FUNCTION_BLOCK AddPermitter (* Composite Function Block Type *)
  (* Standard: 61499-2 *)
  (* Version 0.0, 10/19/2017, chivdan, nxtControl GmbH, template *)
  PACKAGE Main;
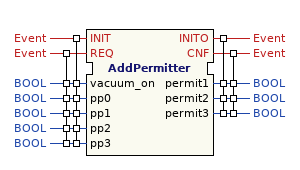
  EVENT_INPUT
    INIT WITH vacuum_on, pp0, pp1, pp2, pp3; (* Initialization Request *)
    REQ WITH vacuum_on, pp0, pp1, pp2, pp3;
  END_EVENT
  EVENT_OUTPUT
    INITO WITH permit1, permit2, permit3; (* Initialization Confirm *)
    CNF WITH permit1, permit2, permit3; (* Execution Confirmation *)
  END_EVENT
  VAR_INPUT
    vacuum_on : BOOL; (* Input event qualifier *)
    pp0 : BOOL;
    pp1 : BOOL;
    pp2 : BOOL;
    pp3 : BOOL;
  END_VAR
  VAR_OUTPUT
    permit1 : BOOL; (* Output event qualifier *)
    permit2 : BOOL;
    permit3 : BOOL;
  END_VAR
  FBS
    WP1 : pickup;
    WP2 : pickup;
    WP3 : pickup;
    FB1 : RandomAddSupplier;
    FB2 : AND_EVENTS;
    FB3 : AND_-2118623424; {SET_ATTRIBUTE(Configuration.GenericFBType.InterfaceParams, Runtime.Standard#CNT:=2;OUT:BOOL)}
    FB4 : AND_EVENTS;
    FB5 : AND_-2118623424; {SET_ATTRIBUTE(Configuration.GenericFBType.InterfaceParams, Runtime.Standard#CNT:=2;OUT:BOOL)}
    FB6 : AND_EVENTS;
    FB7 : AND_-2118623424; {SET_ATTRIBUTE(Configuration.GenericFBType.InterfaceParams, Runtime.Standard#CNT:=2;OUT:BOOL)}
    FB8 : E_MERGE;
    FB9 : E_MERGE;
  END_FBS
  EVENT_CONNECTIONS
    INIT TO WP1.INIT;
    WP1.INITO TO WP2.INIT;
    WP2.INITO TO WP3.INIT;
    WP3.INITO TO INITO;
    INIT TO FB1.INIT;
    FB2.CNF TO FB3.REQ;
    WP1.CNF TO FB2.MODEL;
    FB1.CNF TO FB2.ADDER;
    FB1.CNF TO FB4.ADDER;
    FB1.CNF TO FB6.ADDER;
    WP2.CNF TO FB4.MODEL;
    WP3.CNF TO FB6.MODEL;
    FB4.CNF TO FB5.REQ;
    FB6.CNF TO FB7.REQ;
    FB3.CNF TO FB8.EI1;
    FB5.CNF TO FB8.EI2;
    FB8.EO TO FB9.EI1;
    FB7.CNF TO FB9.EI2;
    FB9.EO TO CNF;
    REQ TO WP1.REQ;
    REQ TO WP2.REQ;
    REQ TO WP3.REQ;
  END_CONNECTIONS
  DATA_CONNECTIONS
    vacuum_on TO WP1.vacuum_on;
    pp1 TO WP1.pp;
    pp2 TO WP2.pp;
    pp3 TO WP3.pp;
    pp0 TO WP1.pp0;
    pp0 TO WP2.pp0;
    pp0 TO WP3.pp0;
    vacuum_on TO WP2.vacuum_on;
    vacuum_on TO WP3.vacuum_on;
    WP1.permit TO FB2.permit;
    FB1.add1 TO FB2.do_add;
    FB2.z1 TO FB3.IN1;
    FB2.z2 TO FB3.IN2;
    FB3.OUT TO permit1;
    WP2.permit TO FB4.permit;
    FB1.add2 TO FB4.do_add;
    WP3.permit TO FB6.permit;
    FB1.add3 TO FB6.do_add;
    FB4.z1 TO FB5.IN1;
    FB4.z2 TO FB5.IN2;
    FB6.z1 TO FB7.IN1;
    FB6.z2 TO FB7.IN2;
    FB5.OUT TO permit2;
    FB7.OUT TO permit3;
  END_CONNECTIONS
END_FUNCTION_BLOCK
